// TIA Portal V18 export
FUNCTION "BoilerActualUnitStatesCtrl" : Void   // FC60108, LAD
{ S7_Optimized_Access := 'TRUE' }
VERSION : 0.1
// Operation Modes                                                 Unit State
// 0=Protection                                                         0=Stopped
// 1=Economy                                                           1=Checking-up  
// 2=PreComfort                                                       2=Preheating
// 3=Comfor                                                              3=Starting 
// 4=Auto(Scheduler)                                              4=RecirculatingOperation
//                                                                                 5=Economy Operation                                                                                                                                            6=PreComfort Operation 
//                                                                                 7=Comfort  operation
//                                                                                 8=Stopping
//                                                                                 9 =Blocking
// stored: AutoNumber false, IsIECCheckEnabled false, SetENOAutomatically false, UDAEnableTagReadback false
   VAR_INPUT
      iUnitID : Int;
      xManualSummer : Bool;
      xManualWinter : Bool;
      cTargetUnitState : Byte;
      cFromHotToColdDelay : Byte;
   END_VAR
   VAR_OUTPUT
      iUnitStateForHMI : Int;
   END_VAR
   VAR_IN_OUT
      cNextUnitState : Byte;
   END_VAR
   VAR_TEMP
      cState : Byte;
   END_VAR
BEGIN

REGION Network 1 (SCL)
   (*
   "BoilerUnitStates".UnitStates.cActual[#iUnitID] = UnitStates.cTarget[iUnitID];
   *)
END_REGION

REGION Network 2 (SCL): Simple state for HMI
END_REGION
END_FUNCTION
